// LS Electric XG5000 project: 과년68_3_3
// PLC NewPLC
// module base 0 slot 0: 입출력 모듈:XBC-DR20S (DC 24V 입력 12점, 릴레이 출력 8점)

PROGRAM NewProgram (task: 스캔 프로그램)

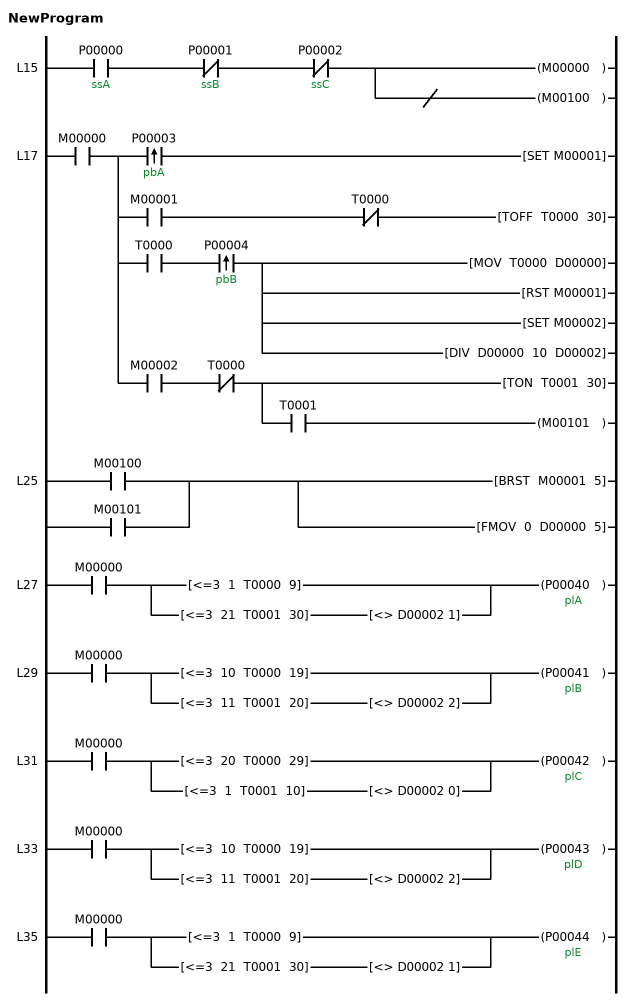
; L15
LOAD      P00000	// ssA
AND NOT   P00001	// ssB
AND NOT   P00002	// ssC
OUT       M00000
NOT
OUT       M00100
; L17
LOAD      M00000
MPUSH
ANDP      P00003	// pbA
SET       M00001
MLOAD
AND       M00001
AND NOT   T0000
TOFF      T0000 30
MLOAD
AND       T0000
ANDP      P00004	// pbB
MOV       T0000 D00000
RST       M00001
SET       M00002
DIV       D00000 10 D00002
MPOP
AND       M00002
AND NOT   T0000
TON       T0001 30
AND       T0001
OUT       M00101
; L25
LOAD      M00100
OR        M00101
BRST      M00001 5
FMOV      0 D00000 5
; L27
LOAD      M00000
LOAD<=3   1 T0000 9
LOAD<=3   21 T0001 30
AND<>     D00002 1
OR LOAD
AND LOAD
OUT       P00040	// plA
; L29
LOAD      M00000
LOAD<=3   10 T0000 19
LOAD<=3   11 T0001 20
AND<>     D00002 2
OR LOAD
AND LOAD
OUT       P00041	// plB
; L31
LOAD      M00000
LOAD<=3   20 T0000 29
LOAD<=3   1 T0001 10
AND<>     D00002 0
OR LOAD
AND LOAD
OUT       P00042	// plC
; L33
LOAD      M00000
LOAD<=3   10 T0000 19
LOAD<=3   11 T0001 20
AND<>     D00002 2
OR LOAD
AND LOAD
OUT       P00043	// plD
; L35
LOAD      M00000
LOAD<=3   1 T0000 9
LOAD<=3   21 T0001 30
AND<>     D00002 1
OR LOAD
AND LOAD
OUT       P00044	// plE

VARIABLES AND COMMENTS (devices not used above)
P00005	BIT	pbC